Fanuc KAREL source: kf00080.KL

-- PROVISIONAL review KL for V770-1; original PC SHA256 fa241c73bf2aa379b50ac9f0555952f4c1e26fab14ea886993204ad2114158aa
-- Incomplete behavior may be omitted. Consult companion uncertainty JSON. Do not deploy.
PROGRAM KF00080
%NOLOCKGROUP
BEGIN
  -- UNRESOLVED_PC offsets 5-15; opcodes 27,22,31
  -- UNRESOLVED_PC offsets 20-24; opcodes 7F
END KF00080
